// TIA Portal V20 export
FUNCTION "LER_PartDataShiftControl" : Void   // FC25, LAD
// stored: Access Published, SetENOAutomatically false
   VAR_INPUT
      shiftCondition : Bool;
      count : Int;
      src_Index : Int;
      dest_Index : Int;
   END_VAR
   VAR_IN_OUT
      PartData : Array[*] of "LER_typePartData";
   END_VAR
   VAR_TEMP
      tempRet_Val : Word;
      tempDeleteData : "LER_typePartData";
   END_VAR
   VAR_TEMP   // added for the SCL form of the ladder/FBD networks
      _w1 : Bool;
   END_VAR
BEGIN

REGION Network 1: Data Shift
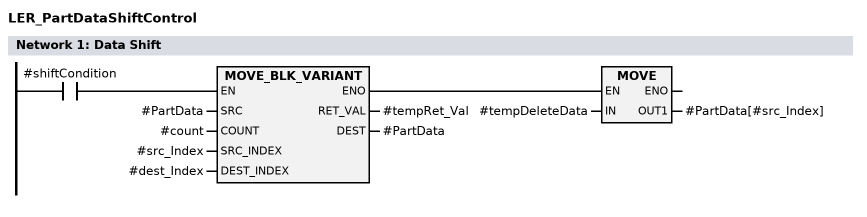
   RUNG wire#powerrail
      Contact( #shiftCondition )
      MOVE_BLK_VARIANT(SRC := #PartData, COUNT := #count, SRC_INDEX := #src_Index, DEST_INDEX := #dest_Index, Ret_Val => #tempRet_Val, DEST => #PartData)
      Move(in := #tempDeleteData, out1 => #PartData[#src_Index])
   END_RUNG
   // the same network as SCL:
   #tempRet_Val := MOVE_BLK_VARIANT(EN := #shiftCondition,
                           SRC := #PartData,
                           COUNT := #count,
                           SRC_INDEX := #src_Index,
                           DEST_INDEX := #dest_Index,
                           DEST => #PartData,
                           ENO => #_w1);
   IF #_w1 THEN #PartData[#src_Index] := #tempDeleteData; END_IF;
END_REGION
END_FUNCTION
